{attribute addProperty BoxType "EK1122-0000-0018"}
{attribute addProperty Id "Beckhoff_ELM3xxx_0030sub_EK1100EK1100_179A0949162"}
{attribute addProperty CRC "2132369187"}
{attribute addProperty SizeInBites "16"}
{attribute addProperty SizeInBytes "2"}
TYPE Beckhoff_ELM3xxx_0030EK1122_7F195F23 EXTENDS EK1122_179A0949 :
STRUCT
	{attribute addProperty Name "Beckhoff_ELM3xxx_0030sub_EK1100"}
	Beckhoff_ELM3xxx_0030sub_EK1100 : EK1100_179A0949;
END_STRUCT
END_TYPE

(* stored: Version 1.2.0.0, ProductVersion 3.1.4024.9
   DUT Beckhoff_ELM3xxx_0030EK1122_7F195F23: Id {d9cfed34-be03-4c5a-a29d-0da3d9145393} *)
